RoboDK station: Tests-Fanuc.rdk

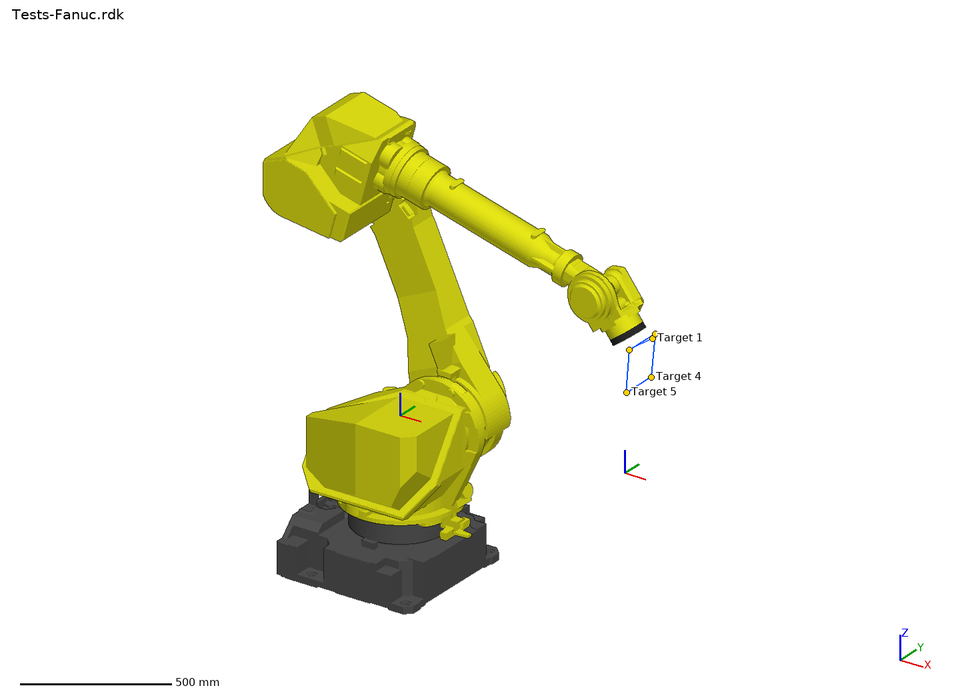
[picture v0: the station drawn from its stored meshes, robots at their saved joint values, targets as dots, program paths as lines]
Station Tests-Fanuc. Poses are relative to the parent item; angles as X-Y-Z fixed-axis rotations.
Station parameters (name, value as stored): IO_5, 1
  - frame Fanuc M-710iC/70 Base at (0, 0, 0) mm
    - robot Fanuc M-710iC/70: 6 axes, payload 70 kg, reach 1360 mm, repeatability 0.07 mm, weight 545 kg
        modified DH rows (alpha deg, a mm, theta deg, d mm): 0, 0, 0, 570; -90, 150, -90, 0; 0, 870, 0, 0; -90, 170, 0, 1016; 90, 0, 0, 0; -90, 0, 0, 175
        base shift (0, 0, -570) mm
        joint limits [-180, -110, -220, -360, -125, -360] to [180, 110, 355, 360, 125, 360]; home [0, 0, 0, 0, 0, 0]; saved at [0, -24.187, -15.328, 0, -37.803, 0]
      - tool Tool, TCP at (-30, 0, 40) mm, rotated rx 0 ry -60 rz 0 deg
    - frame Frame 2 at (904.63, 0, 40.84) mm
      - target Target 1 (joint target) at (113.15, 0, 526.99) mm, rotated rx 180 ry -30 rz 0 deg; joints [0, -24.355, -20.397, -180, -20.397, -180] of Fanuc M-710iC/70
      - target Target 2 (Cartesian target) at (18.72, 0, 458.17) mm, rotated rx -180 ry 23.13 rz 0 deg; joints [0, -3.687, -0.703, 0, -56.115, 0] of Fanuc M-710iC/70
      - target Target 3 (Cartesian target) at (18.72, 147.32, 458.17) mm, rotated rx -180 ry 23.13 rz 0 deg; joints [21.68, 1.512, 4.395, 15.003, -58.895, -25.526] of Fanuc M-710iC/70
      - target Target 4 (Cartesian target) at (3.28, 147.32, 294.99) mm, rotated rx -180 ry 23.13 rz 0 deg; joints [22.53, 1.554, -26.448, 27.261, -30.126, -42.381] of Fanuc M-710iC/70
      - target Target 5 (Cartesian target) at (3.28, 4.68, 294.99) mm, rotated rx -180 ry 23.13 rz 0 deg; joints [0.755, -3.909, -31.79, 1.061, -25.256, -1.564] of Fanuc M-710iC/70
  - program Program (19 instructions, listed below)
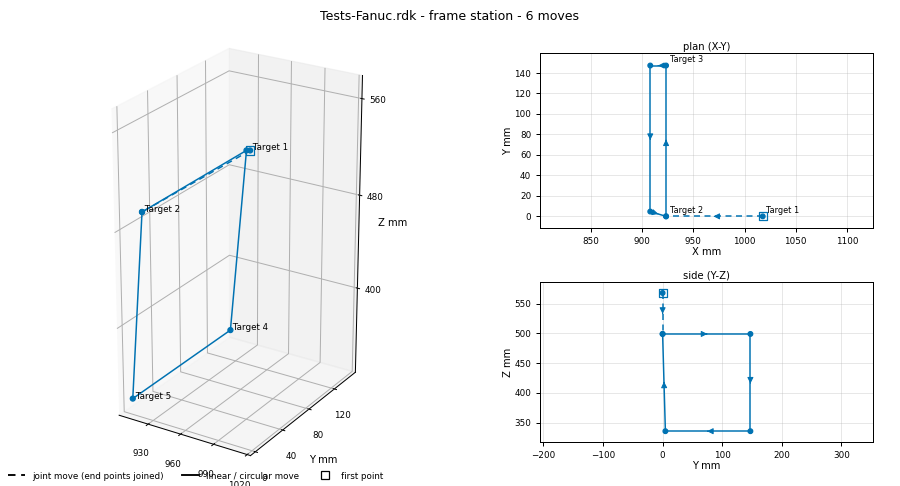
[picture p0: tool path of Tests-Fanuc.rdk in frame station, 6 of 6 moves have a stored position in this frame; points joined in program order, loops and branches not executed]

--- program Program (robot Fanuc M-710iC/70) ---
  Set Ref.: Frame 2
  Set Tool: Tool 1
  Set speed (100.0 mm/s)
  MoveJ (Target 1)
  MoveJ (Target 2)
  Pause 500 ms
  MoveL (Target 3)
  MoveL (Target 4)
  Print: Stop the robot until the user wants to continue
  Remove next line to prevent ...: Remove next line to prevent the robot from stopping
  Stop
  Print: Running program Prog2
  Call Subprog
  MoveL (Target 5)
  Print: Set Digital Output 5 to ON
  Set IO_5=1
  MoveL (Target 2)
  Print: Wait for digital input 5 to turn ON
  Wait IO_5=1
